// Mitsubishi GX Works2 project: 서보_평션_층_20251015   PLC: Q00U

PROGRAM MAIN
VAR
  공급실린더 : CY_W;
  가공실린더 : CY_S;
  송출실린더 : CY_W;
  스토퍼_실린더 : CY_S;
  서보_위치제어 : POS;
  층_위치 : POS;
  흡착실린더 : CY_W;
END_VAR
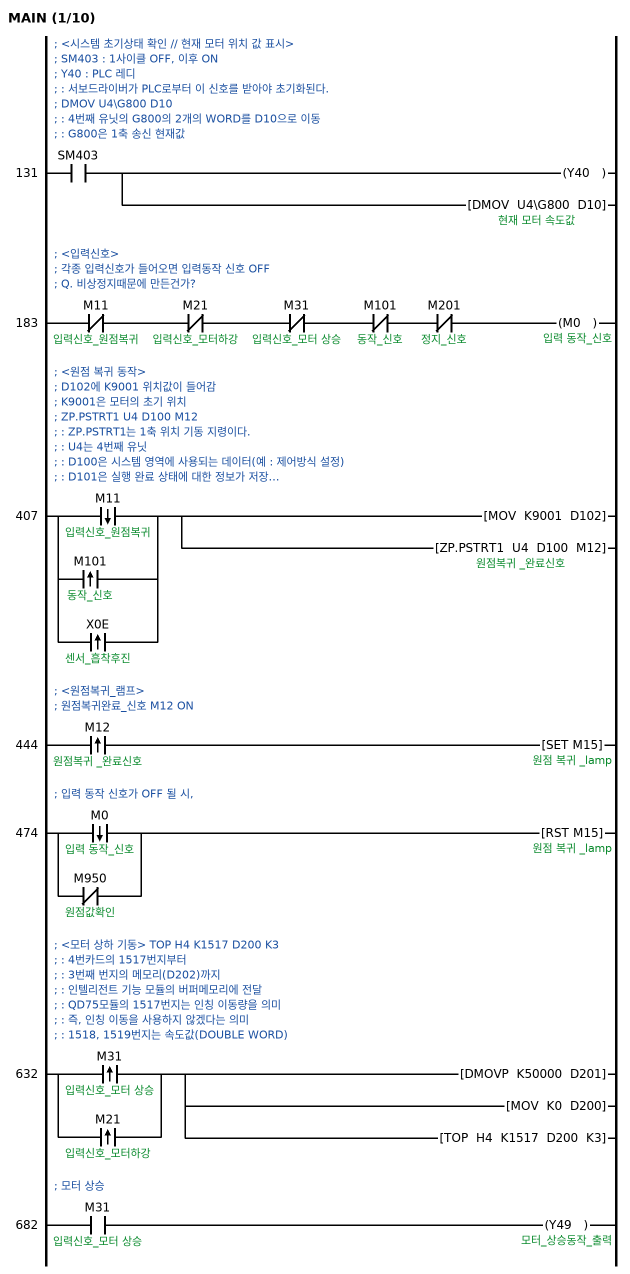
; <시스템 초기상태 확인 // 현재 모터 위치 값 표시>
; SM403 : 1사이클 OFF, 이후 ON
; Y40 : PLC 레디
; : 서보드라이버가 PLC로부터 이 신호를 받아야 초기화된다.
; DMOV U4\G800 D10
; : 4번째 유닛의 G800의 2개의 WORD를 D10으로 이동
; : G800은 1축 송신 현재값
131   LD      SM403
      OUT     Y40
      DMOV    U4\G800 D10  ; 현재 모터 속도값
; <입력신호>
; 각종 입력신호가 들어오면 입력동작 신호 OFF
; Q. 비상정지때문에 만든건가?
183   LDI     M11  ; 입력신호_원점복귀
      ANI     M21  ; 입력신호_모터하강
      ANI     M31  ; 입력신호_모터 상승
      ANI     M101  ; 동작_신호
      ANI     M201  ; 정지_신호
      OUT     M0  ; 입력 동작_신호
; <원점 복귀 동작>
; D102에 K9001 위치값이 들어감
; K9001은 모터의 초기 위치
; ZP.PSTRT1 U4 D100 M12
; : ZP.PSTRT1는 1축 위치 기동 지령이다.
; : U4는 4번째 유닛
; : D100은 시스템 영역에 사용되는 데이터(예 : 제어방식 설정)
; : D101은 실행 완료 상태에 대한 정보가 저장됨
; : D102는 위치 결정 번호
; : ZP.PSTRT1 명령 시작, D100~D102에 저장된 메모리에 따라 기동
; : 기동이 끝나고 정상 완료시, D101 데이터가 0, M12 릴레이 ON
407   LDF     M11  ; 입력신호_원점복귀
      ORP     M101  ; 동작_신호
      ORP     X0E  ; 센서_흡착후진
      MOV     K9001 D102
      ZP.PSTRT1 U4 D100 M12  ; 원점복귀 _완료신호
; <원점복귀_램프>
; 원점복귀완료_신호 M12 ON
444   LDP     M12  ; 원점복귀 _완료신호
      SET     M15  ; 원점 복귀 _lamp
        [note] 원점복귀 램프 M15 ON
; 입력 동작 신호가 OFF 될 시,
474   LDF     M0  ; 입력 동작_신호
      ORI     M950  ; 원점값확인
      RST     M15  ; 원점 복귀 _lamp
        [note] 원점복귀 램프 M15 OFF
; <모터 상하 기동> TOP H4 K1517 D200 K3
; : 4번카드의 1517번지부터
; : 3번째 번지의 메모리(D202)까지
; : 인텔리전트 기능 모듈의 버퍼메모리에 전달
; : QD75모듈의 1517번지는 인칭 이동량을 의미
; : 즉, 인칭 이동을 사용하지 않겠다는 의미
; : 1518, 1519번지는 속도값(DOUBLE WORD)
632   LDP     M31  ; 입력신호_모터 상승
      ORP     M21  ; 입력신호_모터하강
      DMOVP   K50000 D201
        [note] 속도값을 D201~ 메모리로 이동
      MOV     K0 D200
        [note] 0을 D200으로 이동(초기화)
      TOP     H4 K1517 D200 K3
; 모터 상승
682   LD      M31  ; 입력신호_모터 상승
      OUT     Y49  ; 모터_상승동작_출력
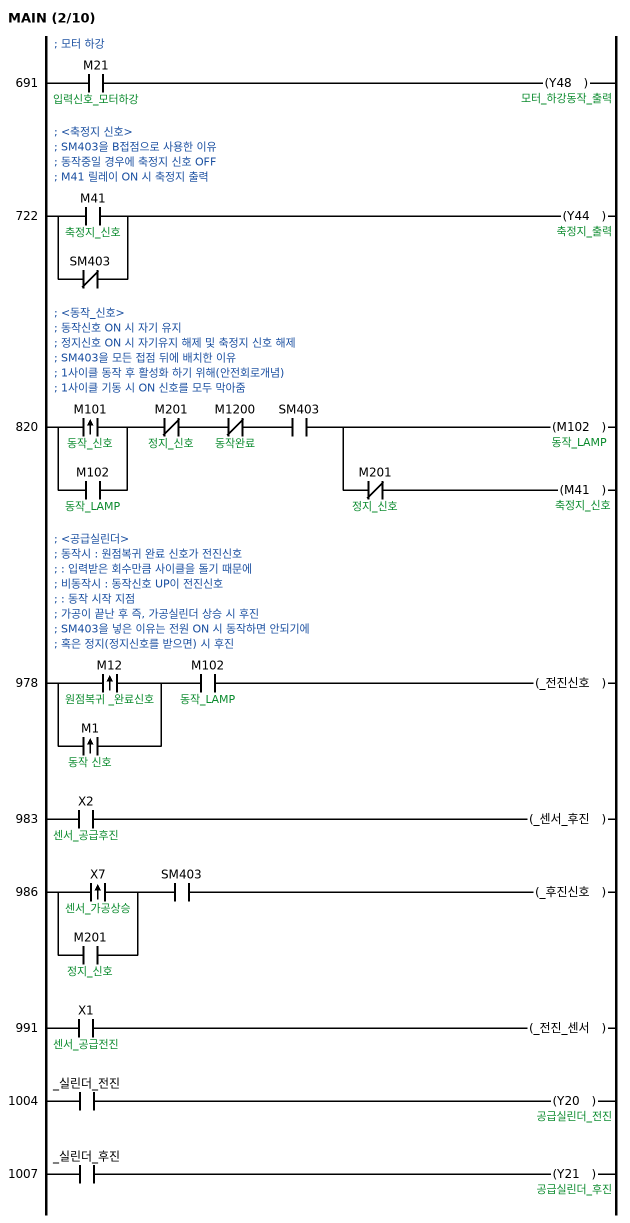
; 모터 하강
691   LD      M21  ; 입력신호_모터하강
      OUT     Y48  ; 모터_하강동작_출력
; <축정지 신호>
; SM403을 B접점으로 사용한 이유
; 동작중일 경우에 축정지 신호 OFF
; M41 릴레이 ON 시 축정지 출력
722   LD      M41  ; 축정지_신호
      ORI     SM403
      OUT     Y44  ; 축정지_출력
; <동작_신호>
; 동작신호 ON 시 자기 유지
; 정지신호 ON 시 자기유지 해제 및 축정지 신호 해제
; SM403을 모든 접점 뒤에 배치한 이유
; 1사이클 동작 후 활성화 하기 위해(안전회로개념)
; 1사이클 기동 시 ON 신호를 모두 막아줌
820   LDP     M101  ; 동작_신호
      OR      M102  ; 동작_LAMP
      ANI     M201  ; 정지_신호
      ANI     M1200  ; 동작완료
      AND     SM403
      OUT     M102  ; 동작_LAMP
      ANI     M201  ; 정지_신호
      OUT     M41  ; 축정지_신호
; FB BLK START CY_W(공급실린더)
; <공급실린더>
; 동작시 : 원점복귀 완료 신호가 전진신호
; : 입력받은 회수만큼 사이클을 돌기 때문에
; 비동작시 : 동작신호 UP이 전진신호
; : 동작 시작 지점
; 가공이 끝난 후 즉, 가공실린더 상승 시 후진
; SM403을 넣은 이유는 전원 ON 시 동작하면 안되기에
; 혹은 정지(정지신호를 받으면) 시 후진
978   LDP     M12  ; 원점복귀 _완료신호
      ORP     M1  ; 동작 신호
      AND     M102  ; 동작_LAMP
      OUT     _전진신호
983   LD      X2  ; 센서_공급후진
      OUT     _센서_후진
986   LDP     X7  ; 센서_가공상승
      OR      M201  ; 정지_신호
      AND     SM403
      OUT     _후진신호
991   LD      X1  ; 센서_공급전진
      OUT     _전진_센서
; FB START
; FB_NAME CY_W
; INSTANCE_NAME 공급실린더
; FB IN_B:전진신호
; FB OUT_실린더_전진:B
; FB IN_B:센서_후진
; FB OUT_실린더_후진:B
; FB IN_B:후진신호
; FB IN_B:전진_센서
; FB END
1004  LD      _실린더_전진
      OUT     Y20  ; 공급실린더_전진
1007  LD      _실린더_후진
      OUT     Y21  ; 공급실린더_후진
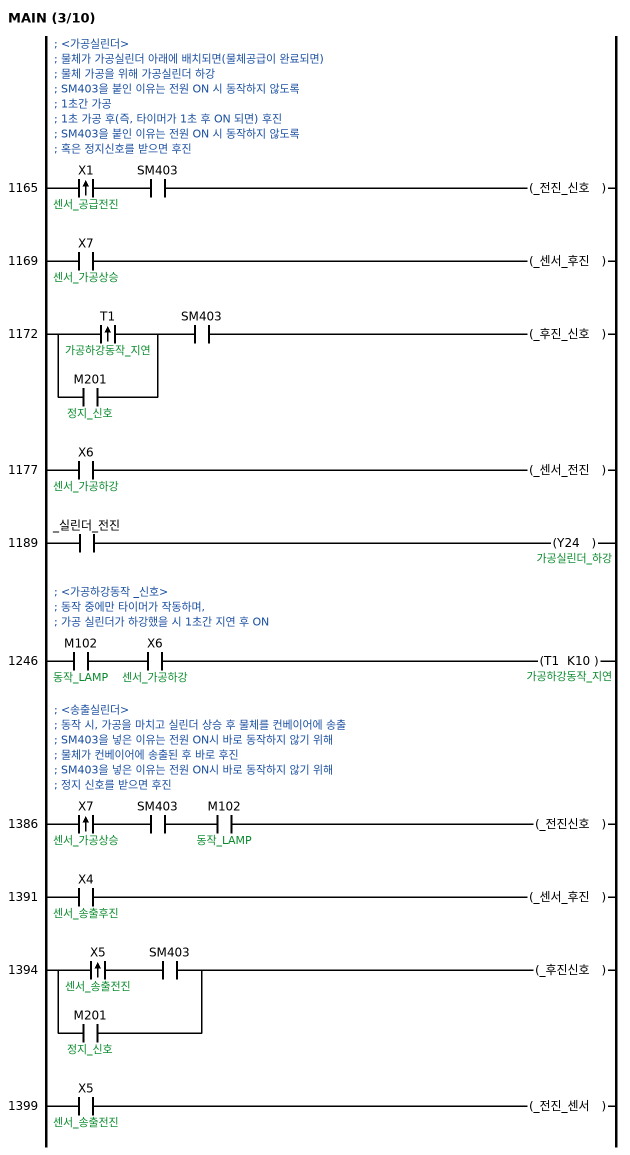
; FB BLK END
; FB BLK START CY_S(가공실린더)
; <가공실린더>
; 물체가 가공실린더 아래에 배치되면(물체공급이 완료되면)
; 물체 가공을 위해 가공실린더 하강
; SM403을 붙인 이유는 전원 ON 시 동작하지 않도록
; 1초간 가공
; 1초 가공 후(즉, 타이머가 1초 후 ON 되면) 후진
; SM403을 붙인 이유는 전원 ON 시 동작하지 않도록
; 혹은 정지신호를 받으면 후진
1165  LDP     X1  ; 센서_공급전진
      AND     SM403
      OUT     _전진_신호
1169  LD      X7  ; 센서_가공상승
      OUT     _센서_후진
1172  LDP     T1  ; 가공하강동작_지연
      OR      M201  ; 정지_신호
      AND     SM403
      OUT     _후진_신호
1177  LD      X6  ; 센서_가공하강
      OUT     _센서_전진
; FB START
; FB_NAME CY_S
; INSTANCE_NAME 가공실린더
; FB IN_B:전진_신호
; FB OUT_실린더_전진:B
; FB IN_B:센서_후진
; FB IN_B:후진_신호
; FB IN_B:센서_전진
; FB END
1189  LD      _실린더_전진
      OUT     Y24  ; 가공실린더_하강
; FB BLK END
; <가공하강동작 _신호>
; 동작 중에만 타이머가 작동하며,
; 가공 실린더가 하강했을 시 1초간 지연 후 ON
1246  LD      M102  ; 동작_LAMP
      AND     X6  ; 센서_가공하강
      OUT     T1 K10  ; 가공하강동작_지연
; FB BLK START CY_W(송출실린더)
; <송출실린더>
; 동작 시, 가공을 마치고 실린더 상승 후 물체를 컨베이어에 송출
; SM403을 넣은 이유는 전원 ON시 바로 동작하지 않기 위해
; 물체가 컨베이어에 송출된 후 바로 후진
; SM403을 넣은 이유는 전원 ON시 바로 동작하지 않기 위해
; 정지 신호를 받으면 후진
1386  LDP     X7  ; 센서_가공상승
      AND     SM403
      AND     M102  ; 동작_LAMP
      OUT     _전진신호
1391  LD      X4  ; 센서_송출후진
      OUT     _센서_후진
1394  LDP     X5  ; 센서_송출전진
      AND     SM403
      OR      M201  ; 정지_신호
      OUT     _후진신호
1399  LD      X5  ; 센서_송출전진
      OUT     _전진_센서
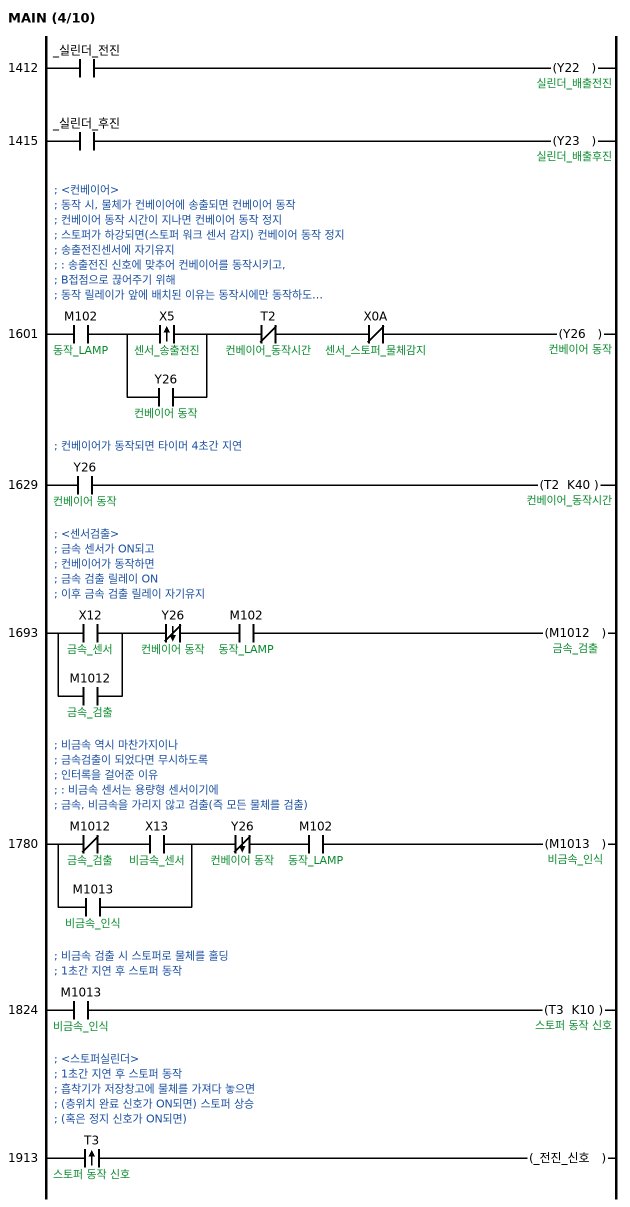
; FB START
; FB_NAME CY_W
; INSTANCE_NAME 송출실린더
; FB IN_B:전진신호
; FB OUT_실린더_전진:B
; FB IN_B:센서_후진
; FB OUT_실린더_후진:B
; FB IN_B:후진신호
; FB IN_B:전진_센서
; FB END
1412  LD      _실린더_전진
      OUT     Y22  ; 실린더_배출전진
1415  LD      _실린더_후진
      OUT     Y23  ; 실린더_배출후진
; FB BLK END
; <컨베이어>
; 동작 시, 물체가 컨베이어에 송출되면 컨베이어 동작
; 컨베이어 동작 시간이 지나면 컨베이어 동작 정지
; 스토퍼가 하강되면(스토퍼 워크 센서 감지) 컨베이어 동작 정지
; 송출전진센서에 자기유지
; : 송출전진 신호에 맞추어 컨베이어를 동작시키고,
; B접점으로 끊어주기 위해
; 동작 릴레이가 앞에 배치된 이유는 동작시에만 동작하도록
; 동작 릴레이는 늘 최우선으로 배치한다.
1601  LD      M102  ; 동작_LAMP
      LDP     X5  ; 센서_송출전진
      OR      Y26  ; 컨베이어 동작
      ANB
      ANI     T2  ; 컨베이어_동작시간
      ANI     X0A  ; 센서_스토퍼_물체감지
      OUT     Y26  ; 컨베이어 동작
; 컨베이어가 동작되면 타이머 4초간 지연
1629  LD      Y26  ; 컨베이어 동작
      OUT     T2 K40  ; 컨베이어_동작시간
; <센서검출>
; 금속 센서가 ON되고
; 컨베이어가 동작하면
; 금속 검출 릴레이 ON
; 이후 금속 검출 릴레이 자기유지
1693  LD      X12  ; 금속_센서
      OR      M1012  ; 금속_검출
      ANDFI   Y26  ; 컨베이어 동작
      AND     M102  ; 동작_LAMP
      OUT     M1012  ; 금속_검출
; 비금속 역시 마찬가지이나
; 금속검출이 되었다면 무시하도록
; 인터록을 걸어준 이유
; : 비금속 센서는 용량형 센서이기에
; 금속, 비금속을 가리지 않고 검출(즉 모든 물체를 검출)
1780  LDI     M1012  ; 금속_검출
      AND     X13  ; 비금속_센서
      OR      M1013  ; 비금속_인식
      ANDFI   Y26  ; 컨베이어 동작
      AND     M102  ; 동작_LAMP
      OUT     M1013  ; 비금속_인식
; 비금속 검출 시 스토퍼로 물체를 홀딩
; 1초간 지연 후 스토퍼 동작
1824  LD      M1013  ; 비금속_인식
      OUT     T3 K10  ; 스토퍼 동작 신호
; FB BLK START CY_S(스토퍼_실린더)
; <스토퍼실린더>
; 1초간 지연 후 스토퍼 동작
; 흡착기가 저장창고에 물체를 가져다 놓으면
; (층위치 완료 신호가 ON되면) 스토퍼 상승
; (혹은 정지 신호가 ON되면)
1913  LDP     T3  ; 스토퍼 동작 신호
      OUT     _전진_신호
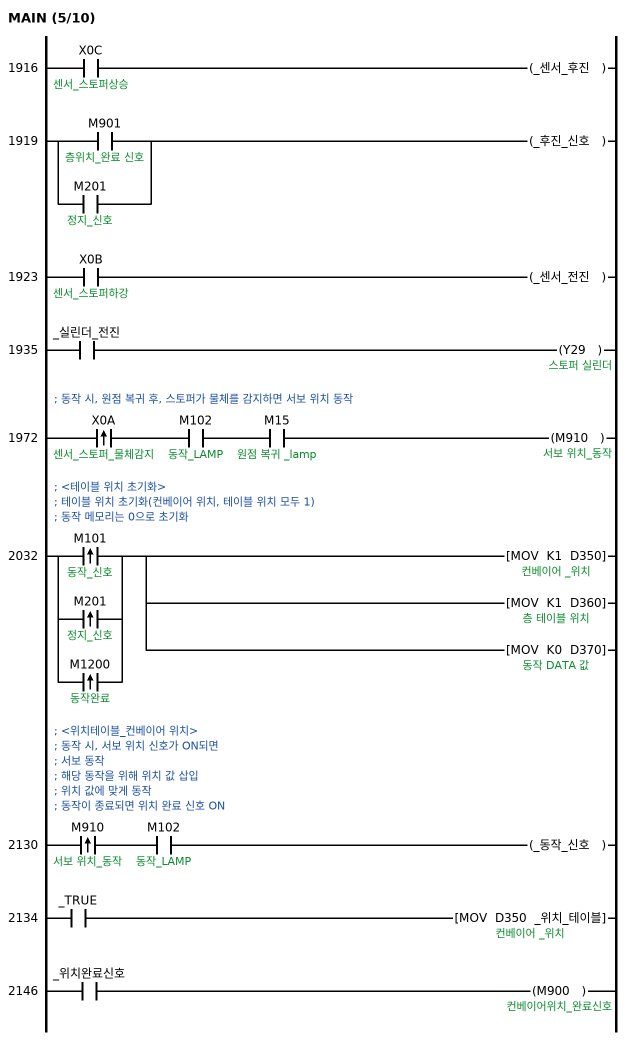
1916  LD      X0C  ; 센서_스토퍼상승
      OUT     _센서_후진
1919  LD      M901  ; 층위치_완료 신호
      OR      M201  ; 정지_신호
      OUT     _후진_신호
1923  LD      X0B  ; 센서_스토퍼하강
      OUT     _센서_전진
; FB START
; FB_NAME CY_S
; INSTANCE_NAME 스토퍼_실린더
; FB IN_B:전진_신호
; FB OUT_실린더_전진:B
; FB IN_B:센서_후진
; FB IN_B:후진_신호
; FB IN_B:센서_전진
; FB END
1935  LD      _실린더_전진
      OUT     Y29  ; 스토퍼 실린더
; FB BLK END
; 동작 시, 원점 복귀 후, 스토퍼가 물체를 감지하면 서보 위치 동작
1972  LDP     X0A  ; 센서_스토퍼_물체감지
      AND     M102  ; 동작_LAMP
      AND     M15  ; 원점 복귀 _lamp
      OUT     M910  ; 서보 위치_동작
; <테이블 위치 초기화>
; 테이블 위치 초기화(컨베이어 위치, 테이블 위치 모두 1)
; 동작 메모리는 0으로 초기화
2032  LDP     M101  ; 동작_신호
      ORP     M201  ; 정지_신호
      ORP     M1200  ; 동작완료
      MOV     K1 D350  ; 컨베이어 _위치
      MOV     K1 D360  ; 층 테이블 위치
      MOV     K0 D370  ; 동작 DATA 값
; FB BLK START POS(서보_위치제어)
; <위치테이블_컨베이어 위치>
; 동작 시, 서보 위치 신호가 ON되면
; 서보 동작
; 해당 동작을 위해 위치 값 삽입
; 위치 값에 맞게 동작
; 동작이 종료되면 위치 완료 신호 ON
2130  LDP     M910  ; 서보 위치_동작
      AND     M102  ; 동작_LAMP
      OUT     _동작_신호
2134  LD      _TRUE
      MOV     D350 _위치_테이블
; FB START
; FB_NAME POS
; INSTANCE_NAME 서보_위치제어
; FB IN_B:동작_신호
; FB OUT_위치완료신호:B
; FB IN_W:위치_테이블
; FB END
2146  LD      _위치완료신호
      OUT     M900  ; 컨베이어위치_완료신호
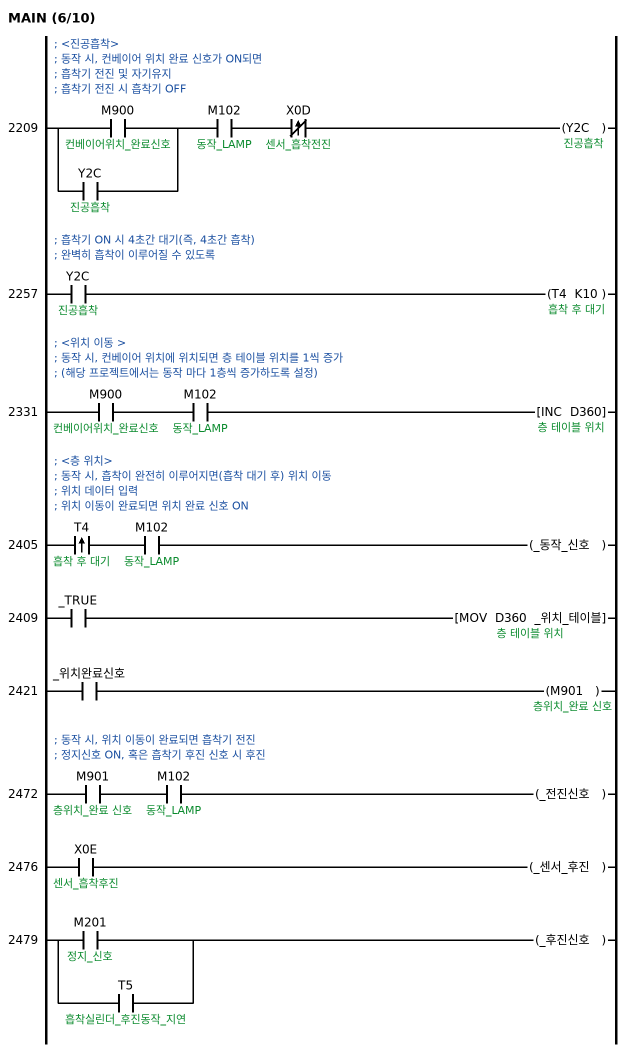
; FB BLK END
; <진공흡착>
; 동작 시, 컨베이어 위치 완료 신호가 ON되면
; 흡착기 전진 및 자기유지
; 흡착기 전진 시 흡착기 OFF
2209  LD      M900  ; 컨베이어위치_완료신호
      OR      Y2C  ; 진공흡착
      AND     M102  ; 동작_LAMP
      ANDPI   X0D  ; 센서_흡착전진
      OUT     Y2C  ; 진공흡착
; 흡착기 ON 시 4초간 대기(즉, 4초간 흡착)
; 완벽히 흡착이 이루어질 수 있도록
2257  LD      Y2C  ; 진공흡착
      OUT     T4 K10  ; 흡착 후 대기
; <위치 이동 >
; 동작 시, 컨베이어 위치에 위치되면 층 테이블 위치를 1씩 증가
; (해당 프로젝트에서는 동작 마다 1층씩 증가하도록 설정)
2331  LD      M900  ; 컨베이어위치_완료신호
      AND     M102  ; 동작_LAMP
      INC     D360
; FB BLK START POS(층_위치)
; <층 위치>
; 동작 시, 흡착이 완전히 이루어지면(흡착 대기 후) 위치 이동
; 위치 데이터 입력
; 위치 이동이 완료되면 위치 완료 신호 ON
2405  LDP     T4  ; 흡착 후 대기
      AND     M102  ; 동작_LAMP
      OUT     _동작_신호
2409  LD      _TRUE
      MOV     D360 _위치_테이블
; FB START
; FB_NAME POS
; INSTANCE_NAME 층_위치
; FB IN_B:동작_신호
; FB OUT_위치완료신호:B
; FB IN_W:위치_테이블
; FB END
2421  LD      _위치완료신호
      OUT     M901  ; 층위치_완료 신호
; FB BLK END
; FB BLK START CY_W(흡착실린더)
; 동작 시, 위치 이동이 완료되면 흡착기 전진
; 정지신호 ON, 혹은 흡착기 후진 신호 시 후진
2472  LD      M901  ; 층위치_완료 신호
      AND     M102  ; 동작_LAMP
      OUT     _전진신호
2476  LD      X0E  ; 센서_흡착후진
      OUT     _센서_후진
2479  LD      M201  ; 정지_신호
      OR      T5  ; 흡착실린더_후진동작_지연
      OUT     _후진신호
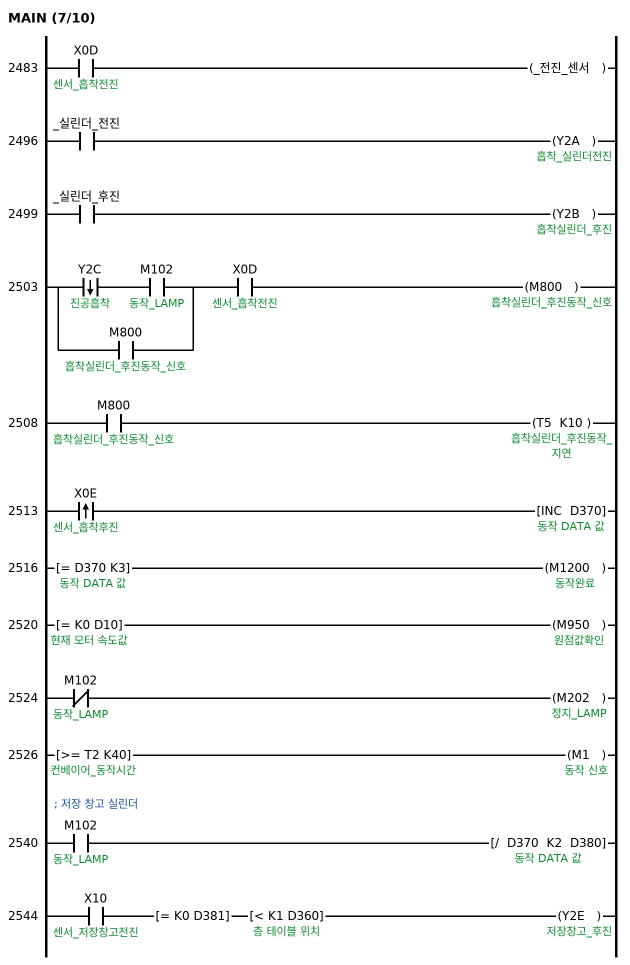
2483  LD      X0D  ; 센서_흡착전진
      OUT     _전진_센서
; FB START
; FB_NAME CY_W
; INSTANCE_NAME 흡착실린더
; FB IN_B:전진신호
; FB OUT_실린더_전진:B
; FB IN_B:센서_후진
; FB OUT_실린더_후진:B
; FB IN_B:후진신호
; FB IN_B:전진_센서
; FB END
2496  LD      _실린더_전진
      OUT     Y2A  ; 흡착_실린더전진
2499  LD      _실린더_후진
      OUT     Y2B  ; 흡착실린더_후진
; FB BLK END
2503  LDF     Y2C  ; 진공흡착
      AND     M102  ; 동작_LAMP
      OR      M800  ; 흡착실린더_후진동작_신호
      AND     X0D  ; 센서_흡착전진
      OUT     M800  ; 흡착실린더_후진동작_신호
2508  LD      M800  ; 흡착실린더_후진동작_신호
      OUT     T5 K10  ; 흡착실린더_후진동작_지연
2513  LDP     X0E  ; 센서_흡착후진
      INC     D370
2516  LD=     D370 K3  ; 동작 DATA 값
      OUT     M1200  ; 동작완료
2520  LD=     K0 D10  ; 현재 모터 속도값
      OUT     M950  ; 원점값확인
2524  LDI     M102  ; 동작_LAMP
      OUT     M202  ; 정지_LAMP
2526  LD>=    T2 K40  ; 컨베이어_동작시간
      OUT     M1  ; 동작 신호
; 저장 창고 실린더
2540  LD      M102  ; 동작_LAMP
      /       D370 K2 D380
2544  LD      X10  ; 센서_저장창고전진
      AND=    K0 D381
      AND<    K1 D360  ; 층 테이블 위치
      OUT     Y2E  ; 저장창고_후진
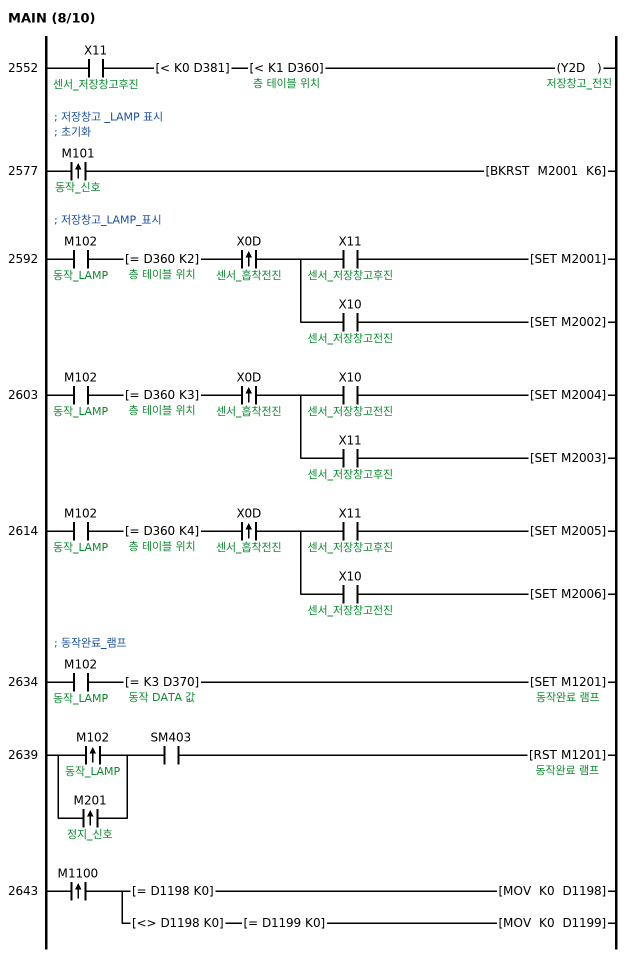
2552  LD      X11  ; 센서_저장창고후진
      AND<    K0 D381
      AND<    K1 D360  ; 층 테이블 위치
      OUT     Y2D  ; 저장창고_전진
; 저장창고 _LAMP 표시
; 초기화
2577  LDP     M101  ; 동작_신호
      BKRST   M2001 K6
; 저장창고_LAMP_표시
2592  LD      M102  ; 동작_LAMP
      AND=    D360 K2  ; 층 테이블 위치
      ANDP    X0D  ; 센서_흡착전진
      MPS
      AND     X11  ; 센서_저장창고후진
      SET     M2001
      MPP
      AND     X10  ; 센서_저장창고전진
      SET     M2002
2603  LD      M102  ; 동작_LAMP
      AND=    D360 K3  ; 층 테이블 위치
      ANDP    X0D  ; 센서_흡착전진
      MPS
      AND     X10  ; 센서_저장창고전진
      SET     M2004
      MPP
      AND     X11  ; 센서_저장창고후진
      SET     M2003
2614  LD      M102  ; 동작_LAMP
      AND=    D360 K4  ; 층 테이블 위치
      ANDP    X0D  ; 센서_흡착전진
      MPS
      AND     X11  ; 센서_저장창고후진
      SET     M2005
      MPP
      AND     X10  ; 센서_저장창고전진
      SET     M2006
; 동작완료_램프
2634  LD      M102  ; 동작_LAMP
      AND=    K3 D370  ; 동작 DATA 값
      SET     M1201  ; 동작완료 램프
2639  LDP     M102  ; 동작_LAMP
      ORP     M201  ; 정지_신호
      AND     SM403
      RST     M1201  ; 동작완료 램프
2643  LDP     M1100
      MPS
      AND=    D1198 K0
      MOV     K0 D1198
      MPP
      AND<>   D1198 K0
      AND=    D1199 K0
      MOV     K0 D1199
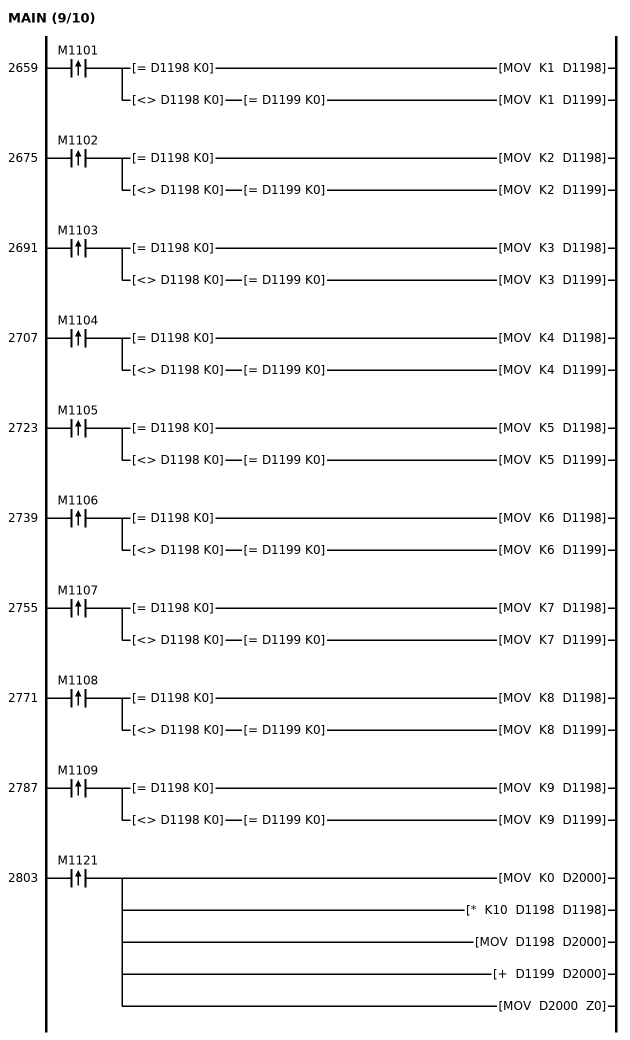
2659  LDP     M1101
      MPS
      AND=    D1198 K0
      MOV     K1 D1198
      MPP
      AND<>   D1198 K0
      AND=    D1199 K0
      MOV     K1 D1199
2675  LDP     M1102
      MPS
      AND=    D1198 K0
      MOV     K2 D1198
      MPP
      AND<>   D1198 K0
      AND=    D1199 K0
      MOV     K2 D1199
2691  LDP     M1103
      MPS
      AND=    D1198 K0
      MOV     K3 D1198
      MPP
      AND<>   D1198 K0
      AND=    D1199 K0
      MOV     K3 D1199
2707  LDP     M1104
      MPS
      AND=    D1198 K0
      MOV     K4 D1198
      MPP
      AND<>   D1198 K0
      AND=    D1199 K0
      MOV     K4 D1199
2723  LDP     M1105
      MPS
      AND=    D1198 K0
      MOV     K5 D1198
      MPP
      AND<>   D1198 K0
      AND=    D1199 K0
      MOV     K5 D1199
2739  LDP     M1106
      MPS
      AND=    D1198 K0
      MOV     K6 D1198
      MPP
      AND<>   D1198 K0
      AND=    D1199 K0
      MOV     K6 D1199
2755  LDP     M1107
      MPS
      AND=    D1198 K0
      MOV     K7 D1198
      MPP
      AND<>   D1198 K0
      AND=    D1199 K0
      MOV     K7 D1199
2771  LDP     M1108
      MPS
      AND=    D1198 K0
      MOV     K8 D1198
      MPP
      AND<>   D1198 K0
      AND=    D1199 K0
      MOV     K8 D1199
2787  LDP     M1109
      MPS
      AND=    D1198 K0
      MOV     K9 D1198
      MPP
      AND<>   D1198 K0
      AND=    D1199 K0
      MOV     K9 D1199
2803  LDP     M1121
      MOV     K0 D2000
      *       K10 D1198 D1198
      MOV     D1198 D2000
      +       D1199 D2000
      MOV     D2000 Z0
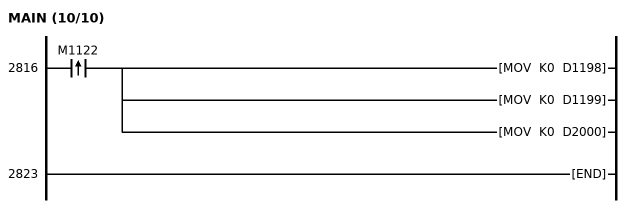
2816  LDP     M1122
      MOV     K0 D1198
      MOV     K0 D1199
      MOV     K0 D2000
2823  END
END_PROGRAM

FUNCTION_BLOCK CY_W
VAR_INPUT
  전진신호 : BOOL;
  센서_후진 : BOOL;
END_VAR
VAR_OUTPUT
  실린더_전진 : BOOL;
END_VAR
VAR_INPUT
  후진신호 : BOOL;
  전진_센서 : BOOL;
END_VAR
VAR_OUTPUT
  실린더_후진 : BOOL;
END_VAR
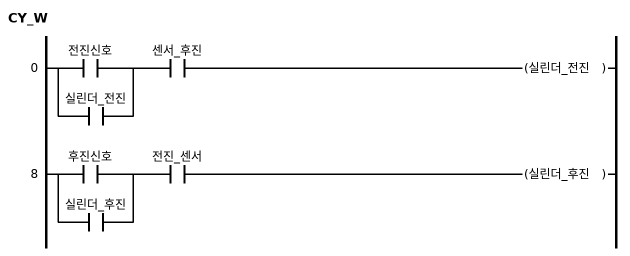
0     LD      전진신호
      OR      실린더_전진
      AND     센서_후진
      OUT     실린더_전진
8     LD      후진신호
      OR      실린더_후진
      AND     전진_센서
      OUT     실린더_후진
END_FUNCTION_BLOCK

FUNCTION_BLOCK CY_S
VAR_INPUT
  전진_신호 : BOOL;
  센서_후진 : BOOL;
END_VAR
VAR
  실린더_후진신호 : BOOL;
END_VAR
VAR_OUTPUT
  실린더_전진 : BOOL;
END_VAR
VAR_INPUT
  후진_신호 : BOOL;
  센서_전진 : BOOL;
END_VAR
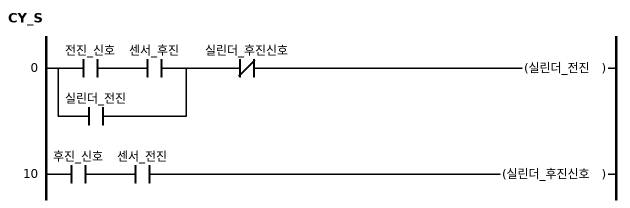
0     LD      전진_신호
      AND     센서_후진
      OR      실린더_전진
      ANI     실린더_후진신호
      OUT     실린더_전진
10    LD      후진_신호
      AND     센서_전진
      OUT     실린더_후진신호
END_FUNCTION_BLOCK

FUNCTION_BLOCK POS
VAR_INPUT
  동작_신호 : BOOL;
  위치_테이블 : INT;
END_VAR
VAR_OUTPUT
  위치완료신호 : BOOL;
END_VAR
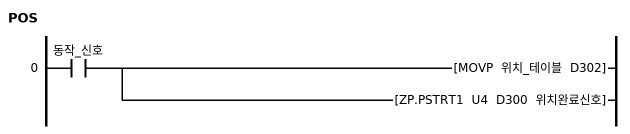
0     LD      동작_신호
      MOVP    위치_테이블 D302
      ZP.PSTRT1 U4 D300 위치완료신호
END_FUNCTION_BLOCK

// device comments not shown above
Y3D  ; 저장창고_전진
M25  ; 하강동작_램프
M35  ; 상승동작_lamp
